// TIA Portal V19 export
FUNCTION_BLOCK "FB_PE_StartStop"   // FB30, FBD
TITLE = Start-stop procedure
{ S7_Optimized_Access := 'FALSE' }
// stored: AutoNumber false, SetENOAutomatically false
   VAR_INPUT
      iCmd_Start : Bool;   // Start command
      iCmd_Stop : Bool;   // Stop command
      iSetting_TON : Time;   // On-delay time for oStarted_TO
      iSetting_TOF : Time;   // Off-delay time for oStarted_TO
   END_VAR
   VAR_OUTPUT
      oStarted : Bool;   // Started signal
      oStarted_TON_TOF : Bool;   // Started with delays signal
   END_VAR
   VAR
      sRE_CmdStart { S7_SetPoint := 'True'} : Bool;
      sStarted { S7_SetPoint := 'True'} : Bool;   // Started not-retain > Automatic restart not allowed during power failures > compliant Machine Directive 2006/42/EG
      sTON_Started { S7_SetPoint := 'True'} : TON_TIME;
      sTOF_Started { S7_SetPoint := 'True'} : TOF_TIME;
   END_VAR
   VAR_TEMP   // added for the SCL form of the ladder/FBD networks
      _w1 : Bool;
   END_VAR
BEGIN

REGION Network 1: Start-stop circuit
   // (**Rising edge on iCmdStart > compliant Machine Directive 2006/42/EG
   // 1) To prevent a reasonably foreseenable human error that could lead to a dangerous situation
   //    Human error = To brigde the start button
   // 2) To prevent that errors in the control logic leads to a dangerous situation
   //    Error in the control logic = Short circuit in the start circuit**)
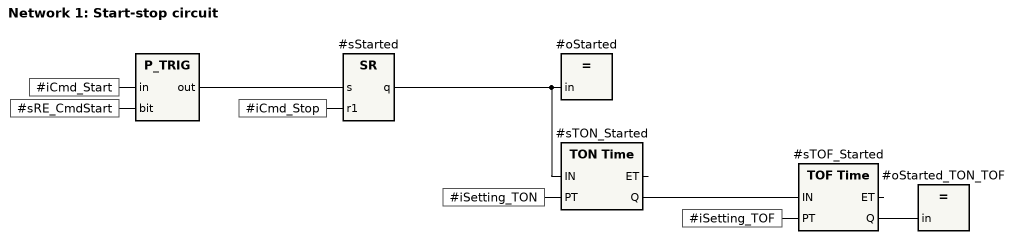
   #_w1 := #iCmd_Start AND NOT #sRE_CmdStart;   // rising edge
   #sRE_CmdStart := #iCmd_Start;
   IF #_w1 THEN
       #sStarted := TRUE;   // SR flip-flop
   END_IF;
   IF #iCmd_Stop THEN #sStarted := FALSE; END_IF;
   #oStarted := #sStarted;
   #sTON_Started(IN := #sStarted, PT := #iSetting_TON);   // TON
   #sTOF_Started(IN := #sTON_Started.Q, PT := #iSetting_TOF);   // TOF
   #oStarted_TON_TOF := #sTOF_Started.Q;
END_REGION
END_FUNCTION_BLOCK
